// TIA Portal V19 export
FUNCTION "FC90_Fault" : Void   // FC90, LAD
{ S7_Optimized_Access := 'TRUE' }
// stored: AutoNumber false, IsIECCheckEnabled true, SetENOAutomatically false
BEGIN

REGION Network 1: Fault no manage by function
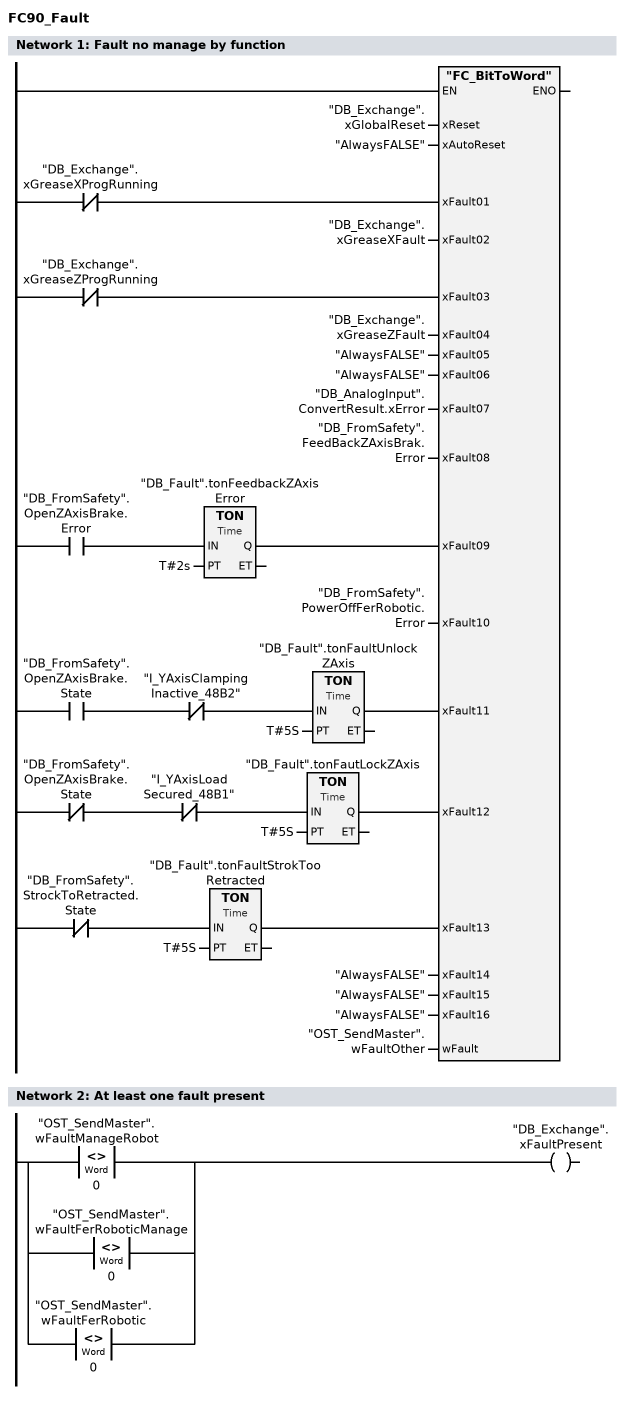
   RUNG wire#powerrail
      "FC_BitToWord"(xFault01 := wire#w1, xFault03 := wire#w2, xFault09 := wire#w3, xFault11 := wire#w4, xFault12 := wire#w5, xFault13 := wire#w6, xReset := "DB_Exchange".xGlobalReset, xAutoReset := "AlwaysFALSE", xFault02 := "DB_Exchange".xGreaseXFault, xFault04 := "DB_Exchange".xGreaseZFault, xFault05 := "AlwaysFALSE", xFault06 := "AlwaysFALSE", xFault07 := "DB_AnalogInput".ConvertResult.xError, xFault08 := "DB_FromSafety".FeedBackZAxisBrak.Error, xFault10 := "DB_FromSafety".PowerOffFerRobotic.Error, xFault14 := "AlwaysFALSE", xFault15 := "AlwaysFALSE", xFault16 := "AlwaysFALSE", wFault := "OST_SendMaster".wFaultOther)
   END_RUNG
   RUNG wire#powerrail
      I_Contact( "DB_Exchange".xGreaseXProgRunning )
   END_RUNG wire#w1
   RUNG wire#powerrail
      I_Contact( "DB_Exchange".xGreaseZProgRunning )
   END_RUNG wire#w2
   RUNG wire#powerrail
      Contact( "DB_FromSafety".OpenZAxisBrake.Error )
      { S7_Templates := "time_type := Time" } "DB_Fault".tonFeedbackZAxisError.TON(pt := T#2s, et =>)
   END_RUNG wire#w3
   RUNG wire#powerrail
      Contact( "DB_FromSafety".OpenZAxisBrake.State )
      I_Contact( "I_YAxisClampingInactive_48B2" )
      { S7_Templates := "time_type := Time" } "DB_Fault".tonFaultUnlockZAxis.TON(pt := T#5S, et =>)
   END_RUNG wire#w4
   RUNG wire#powerrail
      I_Contact( "DB_FromSafety".OpenZAxisBrake.State )
      I_Contact( "I_YAxisLoadSecured_48B1" )
      { S7_Templates := "time_type := Time" } "DB_Fault".tonFautLockZAxis.TON(pt := T#5S, et =>)
   END_RUNG wire#w5
   RUNG wire#powerrail
      I_Contact( "DB_FromSafety".StrockToRetracted.State )
      { S7_Templates := "time_type := Time" } "DB_Fault".tonFaultStrokTooRetracted.TON(pt := T#5S, et =>)
   END_RUNG wire#w6
   // the same network as SCL:
   "DB_Fault".tonFeedbackZAxisError.TON(IN := "DB_FromSafety".OpenZAxisBrake.Error, PT := T#2s);
   "DB_Fault".tonFaultUnlockZAxis.TON(IN := "DB_FromSafety".OpenZAxisBrake.State AND NOT "I_YAxisClampingInactive_48B2",
                           PT := T#5S);
   "DB_Fault".tonFautLockZAxis.TON(IN := NOT "DB_FromSafety".OpenZAxisBrake.State AND NOT "I_YAxisLoadSecured_48B1",
                           PT := T#5S);
   "DB_Fault".tonFaultStrokTooRetracted.TON(IN := NOT "DB_FromSafety".StrockToRetracted.State, PT := T#5S);
   "FC_BitToWord"(xReset := "DB_Exchange".xGlobalReset,
                  xAutoReset := "AlwaysFALSE",
                  xFault01 := NOT "DB_Exchange".xGreaseXProgRunning,
                  xFault02 := "DB_Exchange".xGreaseXFault,
                  xFault03 := NOT "DB_Exchange".xGreaseZProgRunning,
                  xFault04 := "DB_Exchange".xGreaseZFault,
                  xFault05 := "AlwaysFALSE",
                  xFault06 := "AlwaysFALSE",
                  xFault07 := "DB_AnalogInput".ConvertResult.xError,
                  xFault08 := "DB_FromSafety".FeedBackZAxisBrak.Error,
                  xFault09 := "DB_Fault".tonFeedbackZAxisError.Q,
                  xFault10 := "DB_FromSafety".PowerOffFerRobotic.Error,
                  xFault11 := "DB_Fault".tonFaultUnlockZAxis.Q,
                  xFault12 := "DB_Fault".tonFautLockZAxis.Q,
                  xFault13 := "DB_Fault".tonFaultStrokTooRetracted.Q,
                  xFault14 := "AlwaysFALSE",
                  xFault15 := "AlwaysFALSE",
                  xFault16 := "AlwaysFALSE",
                  wFault := "OST_SendMaster".wFaultOther);
END_REGION

REGION Network 2: At least one fault present
   RUNG wire#powerrail
      { S7_Templates := "SrcType := Word" } NE_Contact(in1 := "OST_SendMaster".wFaultManageRobot, in2 := 0)
      wire#w1
      Coil( "DB_Exchange".xFaultPresent )
   END_RUNG
   RUNG wire#powerrail
      { S7_Templates := "SrcType := Word" } NE_Contact(in1 := "OST_SendMaster".wFaultFerRoboticManage, in2 := 0)
   END_RUNG wire#w1
   RUNG wire#powerrail
      { S7_Templates := "SrcType := Word" } NE_Contact(in1 := "OST_SendMaster".wFaultFerRobotic, in2 := 0)
   END_RUNG wire#w1
   // the same network as SCL:
   "DB_Exchange".xFaultPresent := ("OST_SendMaster".wFaultManageRobot <> 0) OR ("OST_SendMaster".wFaultFerRoboticManage <> 0) OR ("OST_SendMaster".wFaultFerRobotic <> 0);
END_REGION
END_FUNCTION
